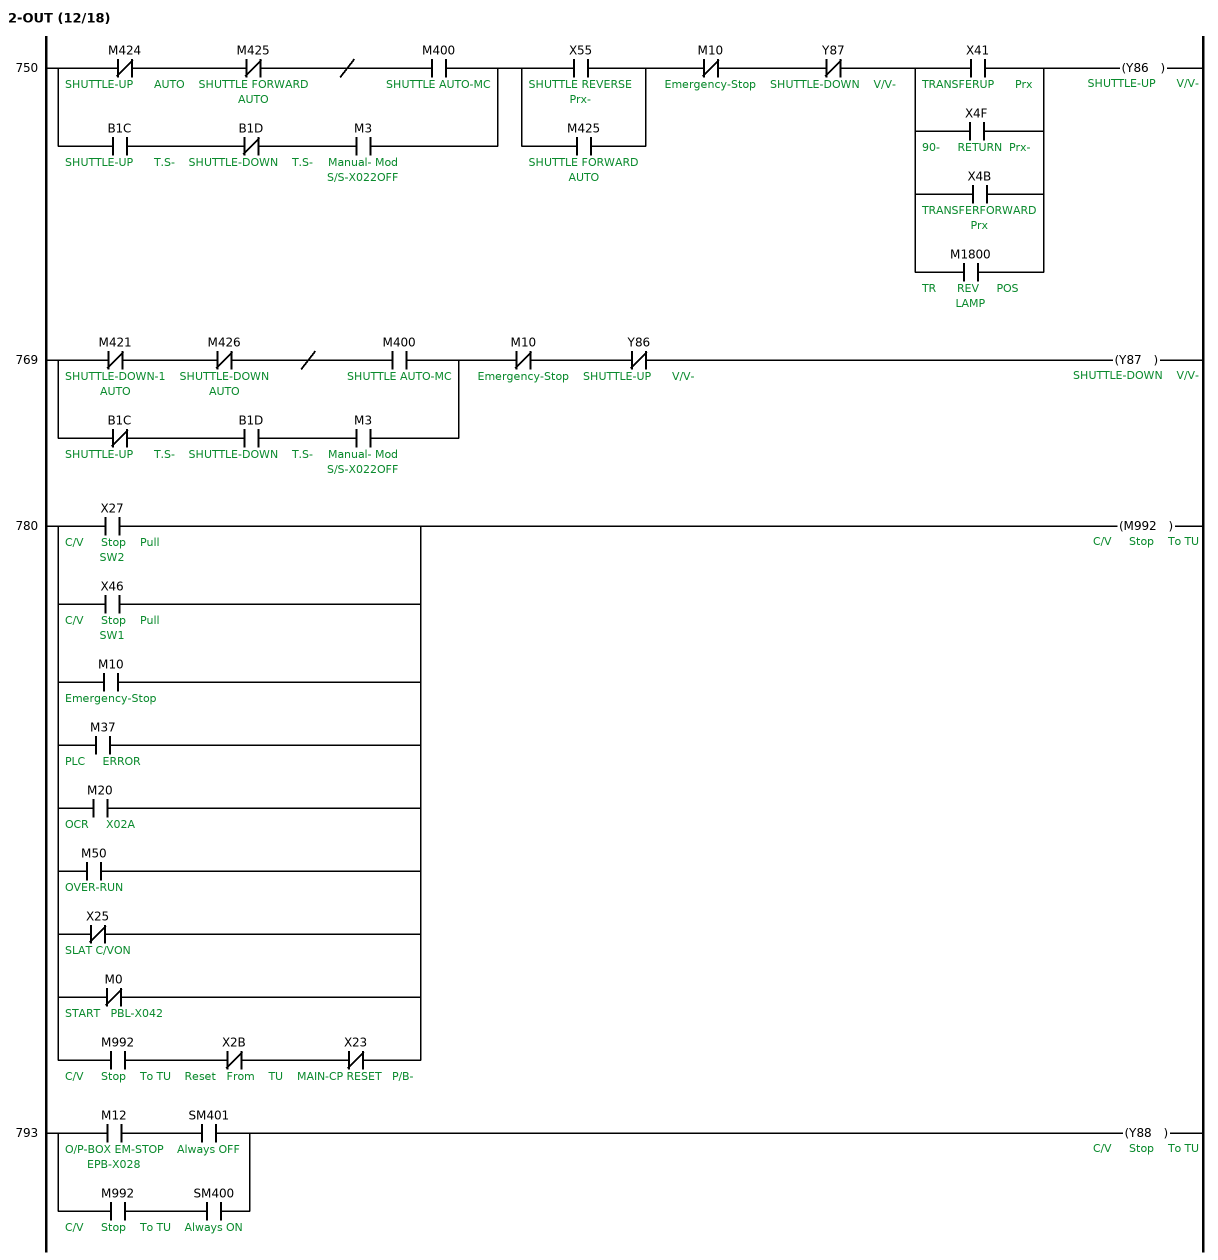
750   LDI     M424  ; SHUTTLE-UP      AUTO
      ANI     M425  ; SHUTTLE FORWARD AUTO
      INV
      AND     M400  ; SHUTTLE AUTO-MC
      LD      B1C  ; SHUTTLE-UP      T.S-
      ANI     B1D  ; SHUTTLE-DOWN    T.S-
      AND     M3  ; Manual- Mod     S/S-X022OFF
      ORB
      LD      X55  ; SHUTTLE REVERSE Prx-
      OR      M425  ; SHUTTLE FORWARD AUTO
      ANB
      ANI     M10  ; Emergency-Stop
      ANI     Y87  ; SHUTTLE-DOWN    V/V-
      LD      X41  ; TRANSFERUP      Prx
      OR      X4F  ; 90-     RETURN  Prx-
      OR      X4B  ; TRANSFERFORWARD Prx
      OR      M1800  ; TR      REV     POS     LAMP
      ANB
      OUT     Y86  ; SHUTTLE-UP      V/V-
769   LDI     M421  ; SHUTTLE-DOWN-1  AUTO
      ANI     M426  ; SHUTTLE-DOWN    AUTO
      INV
      AND     M400  ; SHUTTLE AUTO-MC
      LDI     B1C  ; SHUTTLE-UP      T.S-
      AND     B1D  ; SHUTTLE-DOWN    T.S-
      AND     M3  ; Manual- Mod     S/S-X022OFF
      ORB
      ANI     M10  ; Emergency-Stop
      ANI     Y86  ; SHUTTLE-UP      V/V-
      OUT     Y87  ; SHUTTLE-DOWN    V/V-
780   LD      X27  ; C/V     Stop    Pull    SW2
      OR      X46  ; C/V     Stop    Pull    SW1
      OR      M10  ; Emergency-Stop
      OR      M37  ; PLC     ERROR
      OR      M20  ; OCR     X02A
      OR      M50  ; OVER-RUN
      ORI     X25  ; SLAT C/VON
      ORI     M0  ; START   PBL-X042
      LD      M992  ; C/V     Stop    To TU
      ANI     X2B  ; Reset   From    TU
      ANI     X23  ; MAIN-CP RESET   P/B-
      ORB
      OUT     M992  ; C/V     Stop    To TU
793   LD      M12  ; O/P-BOX EM-STOP EPB-X028
      AND     SM401  ; Always OFF
      LD      M992  ; C/V     Stop    To TU
      AND     SM400  ; Always ON
      ORB
      OUT     Y88  ; C/V     Stop    To TU
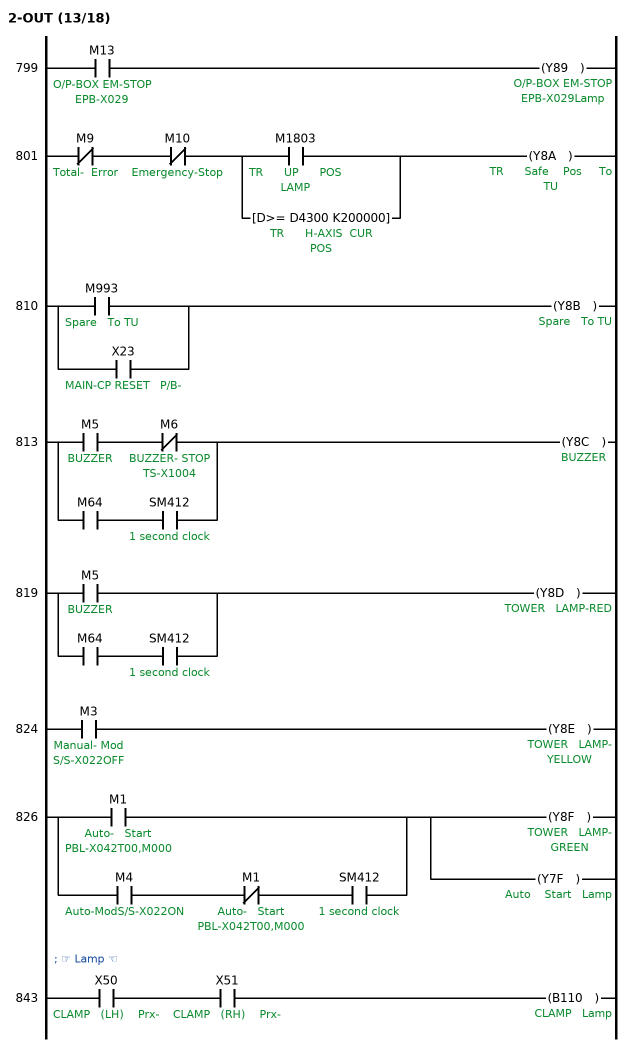
799   LD      M13  ; O/P-BOX EM-STOP EPB-X029
      OUT     Y89  ; O/P-BOX EM-STOP EPB-X029Lamp
801   LDI     M9  ; Total-  Error
      ANI     M10  ; Emergency-Stop
      LD      M1803  ; TR      UP      POS     LAMP
      ORD>=   D4300 K200000  ; TR      H-AXIS  CUR     POS
      ANB
      OUT     Y8A  ; TR      Safe    Pos     To TU
810   LD      M993  ; Spare   To TU
      OR      X23  ; MAIN-CP RESET   P/B-
      OUT     Y8B  ; Spare   To TU
813   LD      M5  ; BUZZER
      ANI     M6  ; BUZZER- STOP    TS-X1004
      LD      M64
      AND     SM412  ; 1 second clock
      ORB
      OUT     Y8C  ; BUZZER
819   LD      M5  ; BUZZER
      LD      M64
      AND     SM412  ; 1 second clock
      ORB
      OUT     Y8D  ; TOWER   LAMP-RED
824   LD      M3  ; Manual- Mod     S/S-X022OFF
      OUT     Y8E  ; TOWER   LAMP-   YELLOW
826   LD      M1  ; Auto-   Start   PBL-X042T00,M000
      LD      M4  ; Auto-ModS/S-X022ON
      ANI     M1  ; Auto-   Start   PBL-X042T00,M000
      AND     SM412  ; 1 second clock
      ORB
      OUT     Y8F  ; TOWER   LAMP-   GREEN
      OUT     Y7F  ; Auto    Start   Lamp
; ☞ Lamp ☜
843   LD      X50  ; CLAMP   (LH)    Prx-
      AND     X51  ; CLAMP   (RH)    Prx-
      OUT     B110  ; CLAMP   Lamp
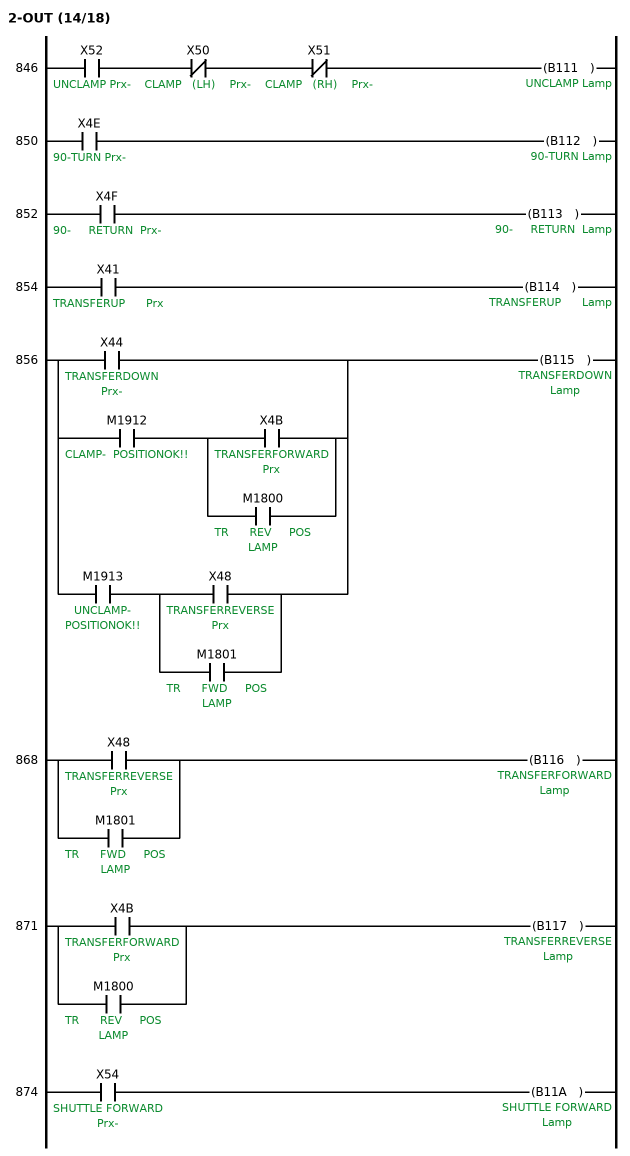
846   LD      X52  ; UNCLAMP Prx-
      ANI     X50  ; CLAMP   (LH)    Prx-
      ANI     X51  ; CLAMP   (RH)    Prx-
      OUT     B111  ; UNCLAMP Lamp
850   LD      X4E  ; 90-TURN Prx-
      OUT     B112  ; 90-TURN Lamp
852   LD      X4F  ; 90-     RETURN  Prx-
      OUT     B113  ; 90-     RETURN  Lamp
854   LD      X41  ; TRANSFERUP      Prx
      OUT     B114  ; TRANSFERUP      Lamp
856   LD      X44  ; TRANSFERDOWN    Prx-
      LD      M1912  ; CLAMP-  POSITIONOK!!
      LD      X4B  ; TRANSFERFORWARD Prx
      OR      M1800  ; TR      REV     POS     LAMP
      ANB
      ORB
      LD      M1913  ; UNCLAMP-POSITIONOK!!
      LD      X48  ; TRANSFERREVERSE Prx
      OR      M1801  ; TR      FWD     POS     LAMP
      ANB
      ORB
      OUT     B115  ; TRANSFERDOWN    Lamp
868   LD      X48  ; TRANSFERREVERSE Prx
      OR      M1801  ; TR      FWD     POS     LAMP
      OUT     B116  ; TRANSFERFORWARD Lamp
871   LD      X4B  ; TRANSFERFORWARD Prx
      OR      M1800  ; TR      REV     POS     LAMP
      OUT     B117  ; TRANSFERREVERSE Lamp
874   LD      X54  ; SHUTTLE FORWARD Prx-
      OUT     B11A  ; SHUTTLE FORWARD Lamp
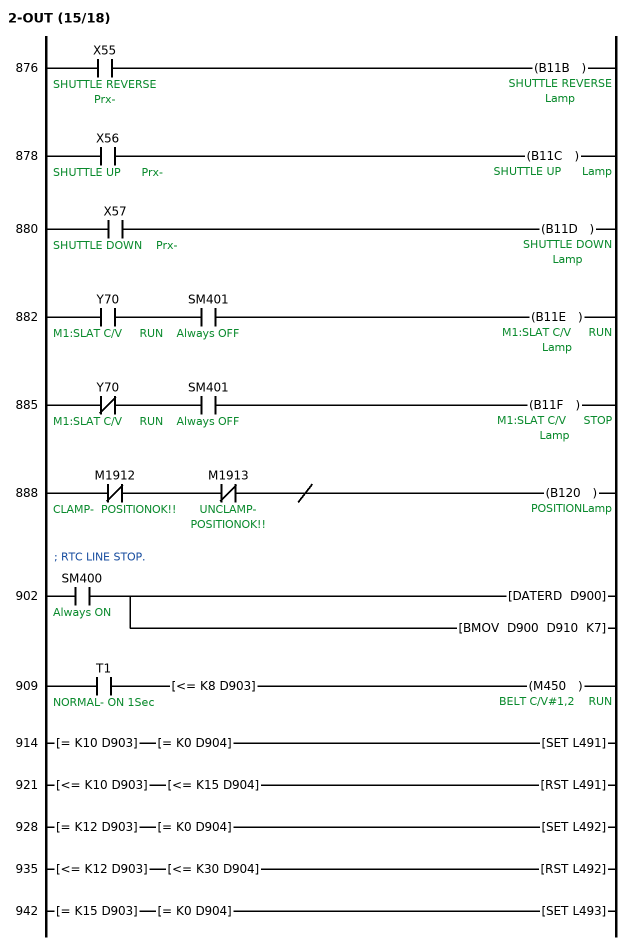
876   LD      X55  ; SHUTTLE REVERSE Prx-
      OUT     B11B  ; SHUTTLE REVERSE Lamp
878   LD      X56  ; SHUTTLE UP      Prx-
      OUT     B11C  ; SHUTTLE UP      Lamp
880   LD      X57  ; SHUTTLE DOWN    Prx-
      OUT     B11D  ; SHUTTLE DOWN    Lamp
882   LD      Y70  ; M1:SLAT C/V     RUN
      AND     SM401  ; Always OFF
      OUT     B11E  ; M1:SLAT C/V     RUN     Lamp
885   LDI     Y70  ; M1:SLAT C/V     RUN
      AND     SM401  ; Always OFF
      OUT     B11F  ; M1:SLAT C/V     STOP    Lamp
888   LDI     M1912  ; CLAMP-  POSITIONOK!!
      ANI     M1913  ; UNCLAMP-POSITIONOK!!
      INV
      OUT     B120  ; POSITIONLamp
; RTC LINE STOP.
902   LD      SM400  ; Always ON
      DATERD  D900
      BMOV    D900 D910 K7
909   LD      T1  ; NORMAL- ON 1Sec
      AND<=   K8 D903
      OUT     M450  ; BELT C/V#1,2    RUN
914   LD=     K10 D903
      AND=    K0 D904
      SET     L491
921   LD<=    K10 D903
      AND<=   K15 D904
      RST     L491
928   LD=     K12 D903
      AND=    K0 D904
      SET     L492
935   LD<=    K12 D903
      AND<=   K30 D904
      RST     L492
942   LD=     K15 D903
      AND=    K0 D904
      SET     L493
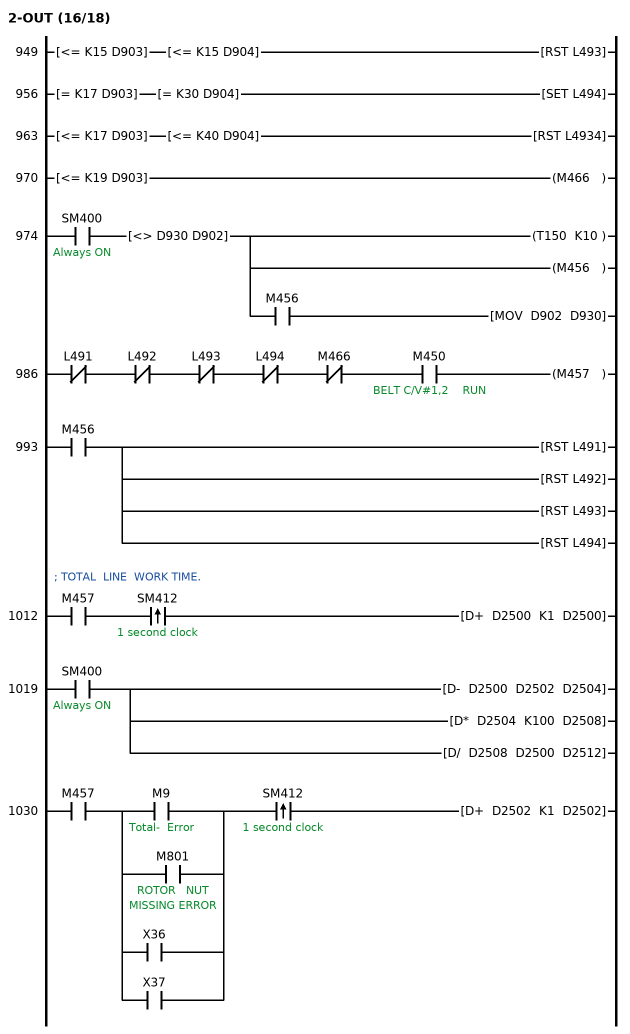
949   LD<=    K15 D903
      AND<=   K15 D904
      RST     L493
956   LD=     K17 D903
      AND=    K30 D904
      SET     L494
963   LD<=    K17 D903
      AND<=   K40 D904
      RST     L4934
970   LD<=    K19 D903
      OUT     M466
974   LD      SM400  ; Always ON
      AND<>   D930 D902
      OUT     T150 K10
      OUT     M456
      AND     M456
      MOV     D902 D930
986   LDI     L491
      ANI     L492
      ANI     L493
      ANI     L494
      ANI     M466
      AND     M450  ; BELT C/V#1,2    RUN
      OUT     M457
993   LD      M456
      RST     L491
      RST     L492
      RST     L493
      RST     L494
; TOTAL  LINE  WORK TIME.
1012  LD      M457
      ANDP    SM412  ; 1 second clock
      D+      D2500 K1 D2500
1019  LD      SM400  ; Always ON
      D-      D2500 D2502 D2504
      D*      D2504 K100 D2508
      D/      D2508 D2500 D2512
1030  LD      M457
      LD      M9  ; Total-  Error
      OR      M801  ; ROTOR   NUT     MISSING ERROR
      OR      X36
      OR      X37
      ANB
      ANDP    SM412  ; 1 second clock
      D+      D2502 K1 D2502
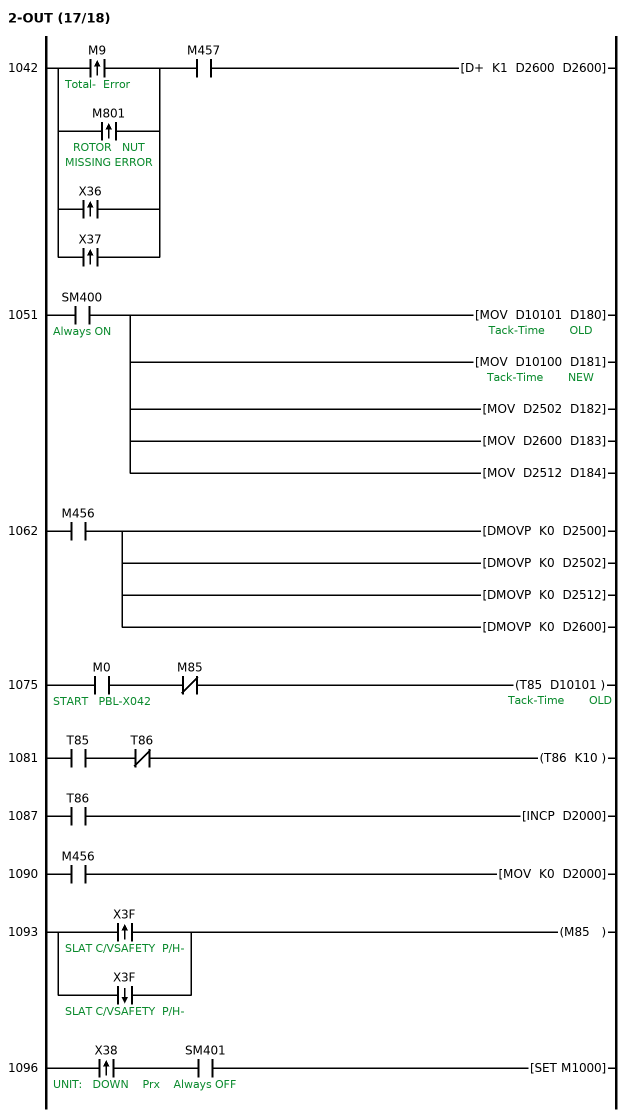
1042  LDP     M9  ; Total-  Error
      ORP     M801  ; ROTOR   NUT     MISSING ERROR
      ORP     X36
      ORP     X37
      AND     M457
      D+      K1 D2600 D2600
1051  LD      SM400  ; Always ON
      MOV     D10101 D180  ; Tack-Time       OLD
      MOV     D10100 D181  ; Tack-Time       NEW
      MOV     D2502 D182
      MOV     D2600 D183
      MOV     D2512 D184
1062  LD      M456
      DMOVP   K0 D2500
      DMOVP   K0 D2502
      DMOVP   K0 D2512
      DMOVP   K0 D2600
1075  LD      M0  ; START   PBL-X042
      ANI     M85
      OUT     T85 D10101  ; Tack-Time       OLD
1081  LD      T85
      ANI     T86
      OUT     T86 K10
1087  LD      T86
      INCP    D2000
1090  LD      M456
      MOV     K0 D2000
1093  LDP     X3F  ; SLAT C/VSAFETY  P/H-
      ORF     X3F  ; SLAT C/VSAFETY  P/H-
      OUT     M85
1096  LDP     X38  ; UNIT:   DOWN    Prx
      AND     SM401  ; Always OFF
      SET     M1000
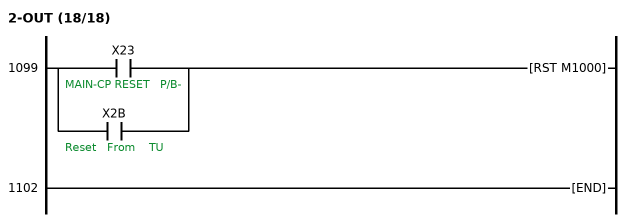
1099  LD      X23  ; MAIN-CP RESET   P/B-
      OR      X2B  ; Reset   From    TU
      RST     M1000
1102  END
END_PROGRAM

PROGRAM 3-ENCORD
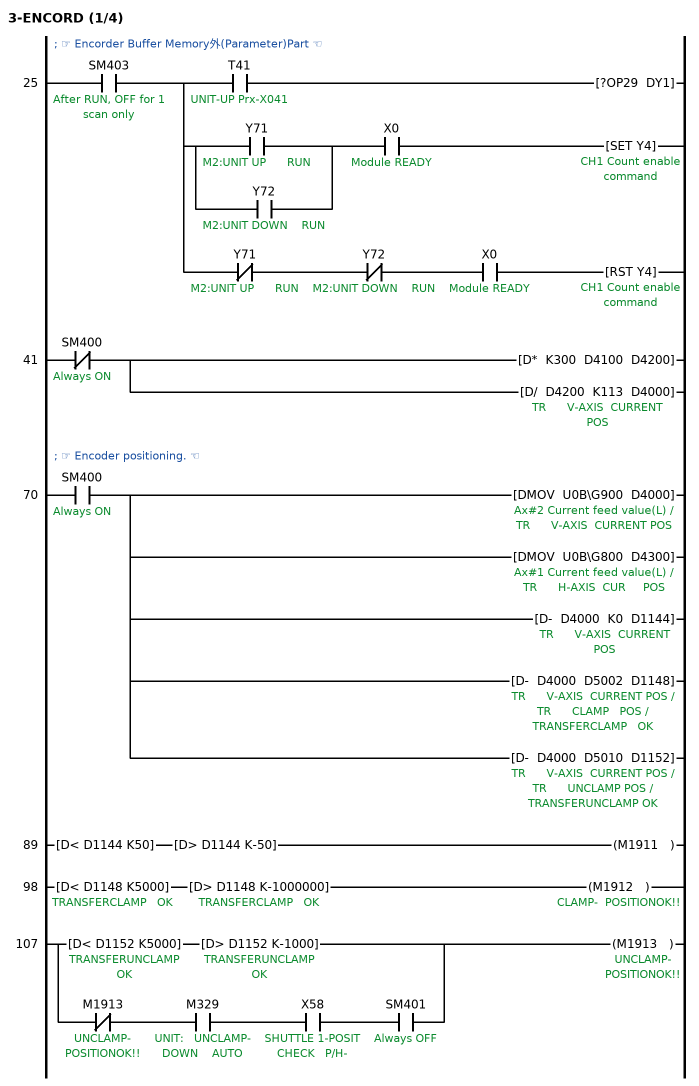
; ☞ Encorder Buffer Memory外(Parameter)Part ☜
25    LD      SM403  ; After RUN, OFF for 1 scan only
      MPS
      AND     T41  ; UNIT-UP Prx-X041
      ?OP29   DY1
      MRD
      LD      Y71  ; M2:UNIT UP      RUN
      OR      Y72  ; M2:UNIT DOWN    RUN
      ANB
      AND     X0  ; Module READY
      SET     Y4  ; CH1 Count enable command
      MPP
      ANI     Y71  ; M2:UNIT UP      RUN
      ANI     Y72  ; M2:UNIT DOWN    RUN
      AND     X0  ; Module READY
      RST     Y4  ; CH1 Count enable command
41    LDI     SM400  ; Always ON
      D*      K300 D4100 D4200
      D/      D4200 K113 D4000  ; TR      V-AXIS  CURRENT POS
; ☞ Encoder positioning. ☜
70    LD      SM400  ; Always ON
      DMOV    U0B\G900 D4000  ; Ax#2 Current feed value(L)
      DMOV    U0B\G800 D4300  ; Ax#1 Current feed value(L) / TR      H-AXIS  CUR     POS
      D-      D4000 K0 D1144
      D-      D4000 D5002 D1148  ; TR      CLAMP   POS / TRANSFERCLAMP   OK
      D-      D4000 D5010 D1152  ; TR      UNCLAMP POS / TRANSFERUNCLAMP OK
89    LDD<    D1144 K50
      ANDD>   D1144 K-50
      OUT     M1911
98    LDD<    D1148 K5000  ; TRANSFERCLAMP   OK
      ANDD>   D1148 K-1000000  ; TRANSFERCLAMP   OK
      OUT     M1912  ; CLAMP-  POSITIONOK!!
107   LDD<    D1152 K5000  ; TRANSFERUNCLAMP OK
      ANDD>   D1152 K-1000  ; TRANSFERUNCLAMP OK
      LDI     M1913  ; UNCLAMP-POSITIONOK!!
      AND     M329  ; UNIT:   UNCLAMP-DOWN    AUTO
      AND     X58  ; SHUTTLE 1-POSIT CHECK   P/H-
      AND     SM401  ; Always OFF
      ORB
      OUT     M1913  ; UNCLAMP-POSITIONOK!!
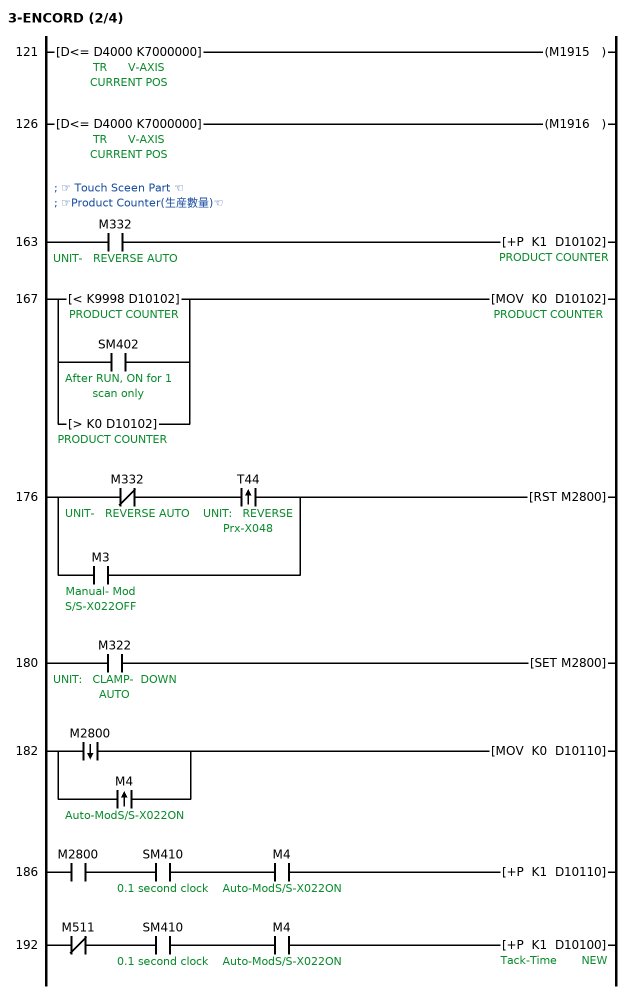
121   LDD<=   D4000 K7000000  ; TR      V-AXIS  CURRENT POS
      OUT     M1915
126   LDD<=   D4000 K7000000  ; TR      V-AXIS  CURRENT POS
      OUT     M1916
; ☞ Touch Sceen Part ☜
; ☞Product Counter(生産數量)☜
163   LD      M332  ; UNIT-   REVERSE AUTO
      +P      K1 D10102  ; PRODUCT COUNTER
167   LD<     K9998 D10102  ; PRODUCT COUNTER
      OR      SM402  ; After RUN, ON for 1 scan only
      OR>     K0 D10102  ; PRODUCT COUNTER
      MOV     K0 D10102
176   LDI     M332  ; UNIT-   REVERSE AUTO
      ANDP    T44  ; UNIT:   REVERSE Prx-X048
      OR      M3  ; Manual- Mod     S/S-X022OFF
      RST     M2800
180   LD      M322  ; UNIT:   CLAMP-  DOWN    AUTO
      SET     M2800
182   LDF     M2800
      ORP     M4  ; Auto-ModS/S-X022ON
      MOV     K0 D10110
186   LD      M2800
      AND     SM410  ; 0.1 second clock
      AND     M4  ; Auto-ModS/S-X022ON
      +P      K1 D10110
192   LDI     M511
      AND     SM410  ; 0.1 second clock
      AND     M4  ; Auto-ModS/S-X022ON
      +P      K1 D10100  ; Tack-Time       NEW
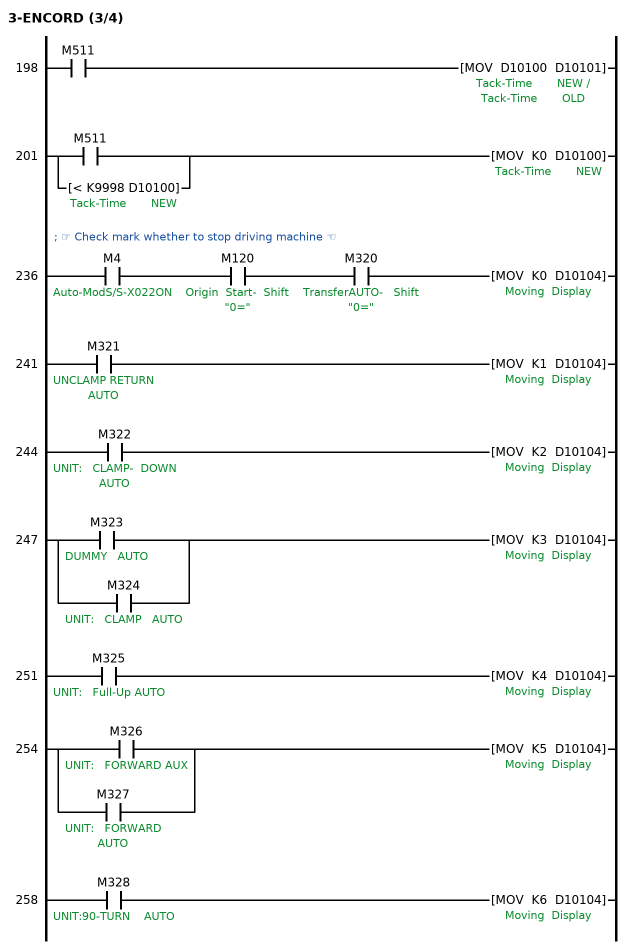
198   LD      M511
      MOV     D10100 D10101  ; Tack-Time       OLD
201   LD      M511
      OR<     K9998 D10100  ; Tack-Time       NEW
      MOV     K0 D10100
; ☞ Check mark whether to stop driving machine ☜
236   LD      M4  ; Auto-ModS/S-X022ON
      AND     M120  ; Origin  Start-  Shift   "0="
      AND     M320  ; TransferAUTO-   Shift   "0="
      MOV     K0 D10104  ; Moving  Display
241   LD      M321  ; UNCLAMP RETURN  AUTO
      MOV     K1 D10104
244   LD      M322  ; UNIT:   CLAMP-  DOWN    AUTO
      MOV     K2 D10104
247   LD      M323  ; DUMMY   AUTO
      OR      M324  ; UNIT:   CLAMP   AUTO
      MOV     K3 D10104
251   LD      M325  ; UNIT:   Full-Up AUTO
      MOV     K4 D10104
254   LD      M326  ; UNIT:   FORWARD AUX
      OR      M327  ; UNIT:   FORWARD AUTO
      MOV     K5 D10104
258   LD      M328  ; UNIT:90-TURN    AUTO
      MOV     K6 D10104
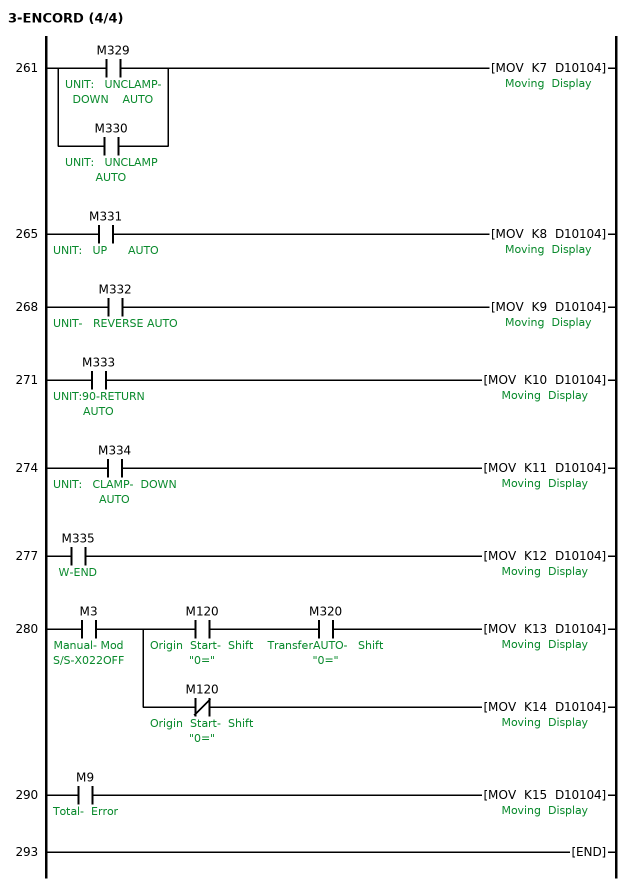
261   LD      M329  ; UNIT:   UNCLAMP-DOWN    AUTO
      OR      M330  ; UNIT:   UNCLAMP AUTO
      MOV     K7 D10104
265   LD      M331  ; UNIT:   UP      AUTO
      MOV     K8 D10104
268   LD      M332  ; UNIT-   REVERSE AUTO
      MOV     K9 D10104
271   LD      M333  ; UNIT:90-RETURN  AUTO
      MOV     K10 D10104
274   LD      M334  ; UNIT:   CLAMP-  DOWN    AUTO
      MOV     K11 D10104
277   LD      M335  ; W-END
      MOV     K12 D10104
280   LD      M3  ; Manual- Mod     S/S-X022OFF
      MPS
      AND     M120  ; Origin  Start-  Shift   "0="
      AND     M320  ; TransferAUTO-   Shift   "0="
      MOV     K13 D10104
      MPP
      ANI     M120  ; Origin  Start-  Shift   "0="
      MOV     K14 D10104
290   LD      M9  ; Total-  Error
      MOV     K15 D10104
293   END
END_PROGRAM

PROGRAM 4-MODEL
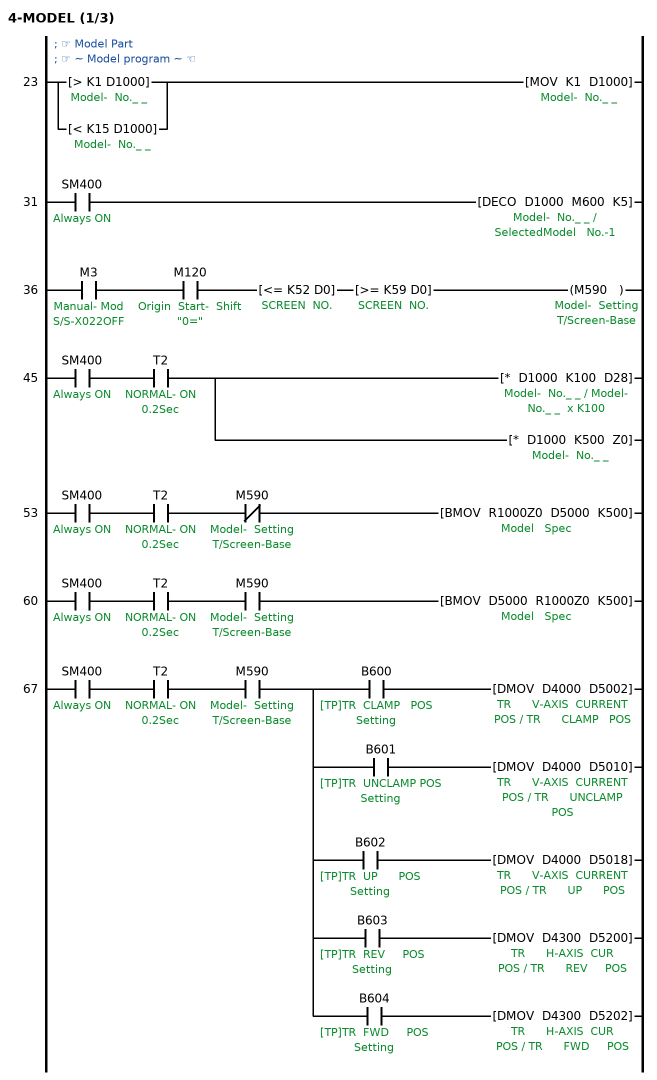
; ☞ Model Part
; ☞ ~ Model program ~ ☜
23    LD>     K1 D1000  ; Model-  No._ _
      OR<     K15 D1000  ; Model-  No._ _
      MOV     K1 D1000
31    LD      SM400  ; Always ON
      DECO    D1000 M600 K5  ; SelectedModel   No.-1
36    LD      M3  ; Manual- Mod     S/S-X022OFF
      AND     M120  ; Origin  Start-  Shift   "0="
      AND<=   K52 D0  ; SCREEN  NO.
      AND>=   K59 D0  ; SCREEN  NO.
      OUT     M590  ; Model-  Setting T/Screen-Base
45    LD      SM400  ; Always ON
      AND     T2  ; NORMAL- ON      0.2Sec
      *       D1000 K100 D28  ; Model-  No._ _  x K100
      *       D1000 K500 Z0
53    LD      SM400  ; Always ON
      AND     T2  ; NORMAL- ON      0.2Sec
      ANI     M590  ; Model-  Setting T/Screen-Base
      BMOV    R1000Z0 D5000 K500  ; Model   Spec
60    LD      SM400  ; Always ON
      AND     T2  ; NORMAL- ON      0.2Sec
      AND     M590  ; Model-  Setting T/Screen-Base
      BMOV    D5000 R1000Z0 K500
67    LD      SM400  ; Always ON
      AND     T2  ; NORMAL- ON      0.2Sec
      AND     M590  ; Model-  Setting T/Screen-Base
      MPS
      AND     B600  ; [TP]TR  CLAMP   POS     Setting
      DMOV    D4000 D5002  ; TR      V-AXIS  CURRENT POS / TR      CLAMP   POS
      MRD
      AND     B601  ; [TP]TR  UNCLAMP POS     Setting
      DMOV    D4000 D5010  ; TR      UNCLAMP POS
      MRD
      AND     B602  ; [TP]TR  UP      POS     Setting
      DMOV    D4000 D5018  ; TR      UP      POS
      MRD
      AND     B603  ; [TP]TR  REV     POS     Setting
      DMOV    D4300 D5200  ; TR      H-AXIS  CUR     POS / TR      REV     POS
      MPP
      AND     B604  ; [TP]TR  FWD     POS     Setting
      DMOV    D4300 D5202  ; TR      FWD     POS
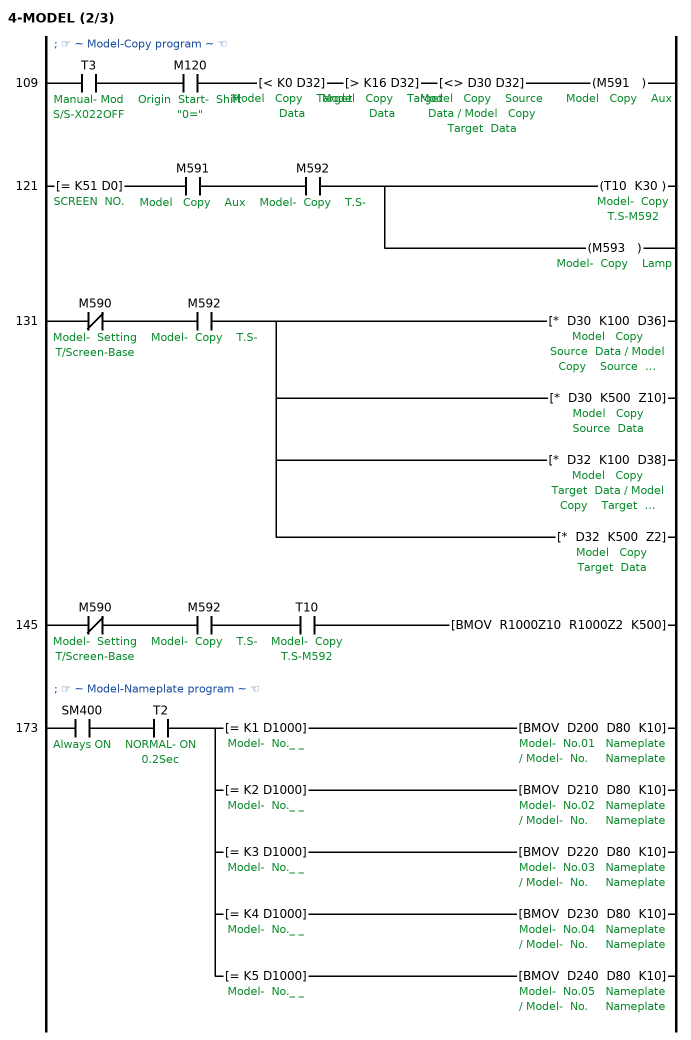
; ☞ ~ Model-Copy program ~ ☜
109   LD      T3  ; Manual- Mod     S/S-X022OFF
      AND     M120  ; Origin  Start-  Shift   "0="
      AND<    K0 D32  ; Model   Copy    Target  Data
      AND>    K16 D32  ; Model   Copy    Target  Data
      AND<>   D30 D32  ; Model   Copy    Source  Data / Model   Copy    Target  Data
      OUT     M591  ; Model   Copy    Aux
121   LD=     K51 D0  ; SCREEN  NO.
      AND     M591  ; Model   Copy    Aux
      AND     M592  ; Model-  Copy    T.S-
      OUT     T10 K30  ; Model-  Copy    T.S-M592
      OUT     M593  ; Model-  Copy    Lamp
131   LDI     M590  ; Model-  Setting T/Screen-Base
      AND     M592  ; Model-  Copy    T.S-
      *       D30 K100 D36  ; Model   Copy    Source  * K100
      *       D30 K500 Z10
      *       D32 K100 D38  ; Model   Copy    Target  * K100
      *       D32 K500 Z2
145   LDI     M590  ; Model-  Setting T/Screen-Base
      AND     M592  ; Model-  Copy    T.S-
      AND     T10  ; Model-  Copy    T.S-M592
      BMOV    R1000Z10 R1000Z2 K500
; ☞ ~ Model-Nameplate program ~ ☜
173   LD      SM400  ; Always ON
      AND     T2  ; NORMAL- ON      0.2Sec
      MPS
      AND=    K1 D1000  ; Model-  No._ _
      BMOV    D200 D80 K10  ; Model-  No.01   Nameplate / Model-  No.     Nameplate
      MRD
      AND=    K2 D1000  ; Model-  No._ _
      BMOV    D210 D80 K10  ; Model-  No.02   Nameplate
      MRD
      AND=    K3 D1000  ; Model-  No._ _
      BMOV    D220 D80 K10  ; Model-  No.03   Nameplate
      MRD
      AND=    K4 D1000  ; Model-  No._ _
      BMOV    D230 D80 K10  ; Model-  No.04   Nameplate
      MPP
      AND=    K5 D1000  ; Model-  No._ _
      BMOV    D240 D80 K10  ; Model-  No.05   Nameplate
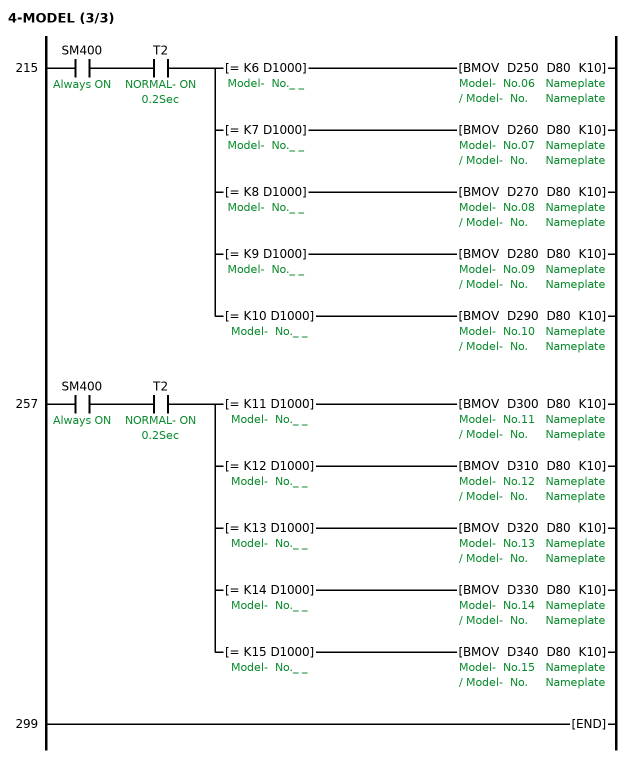
215   LD      SM400  ; Always ON
      AND     T2  ; NORMAL- ON      0.2Sec
      MPS
      AND=    K6 D1000  ; Model-  No._ _
      BMOV    D250 D80 K10  ; Model-  No.06   Nameplate
      MRD
      AND=    K7 D1000  ; Model-  No._ _
      BMOV    D260 D80 K10  ; Model-  No.07   Nameplate
      MRD
      AND=    K8 D1000  ; Model-  No._ _
      BMOV    D270 D80 K10  ; Model-  No.08   Nameplate
      MRD
      AND=    K9 D1000  ; Model-  No._ _
      BMOV    D280 D80 K10  ; Model-  No.09   Nameplate
      MPP
      AND=    K10 D1000  ; Model-  No._ _
      BMOV    D290 D80 K10  ; Model-  No.10   Nameplate
257   LD      SM400  ; Always ON
      AND     T2  ; NORMAL- ON      0.2Sec
      MPS
      AND=    K11 D1000  ; Model-  No._ _
      BMOV    D300 D80 K10  ; Model-  No.11   Nameplate
      MRD
      AND=    K12 D1000  ; Model-  No._ _
      BMOV    D310 D80 K10  ; Model-  No.12   Nameplate
      MRD
      AND=    K13 D1000  ; Model-  No._ _
      BMOV    D320 D80 K10  ; Model-  No.13   Nameplate
      MRD
      AND=    K14 D1000  ; Model-  No._ _
      BMOV    D330 D80 K10  ; Model-  No.14   Nameplate
      MPP
      AND=    K15 D1000  ; Model-  No._ _
      BMOV    D340 D80 K10  ; Model-  No.15   Nameplate
299   END
END_PROGRAM

PROGRAM 5-ERROR
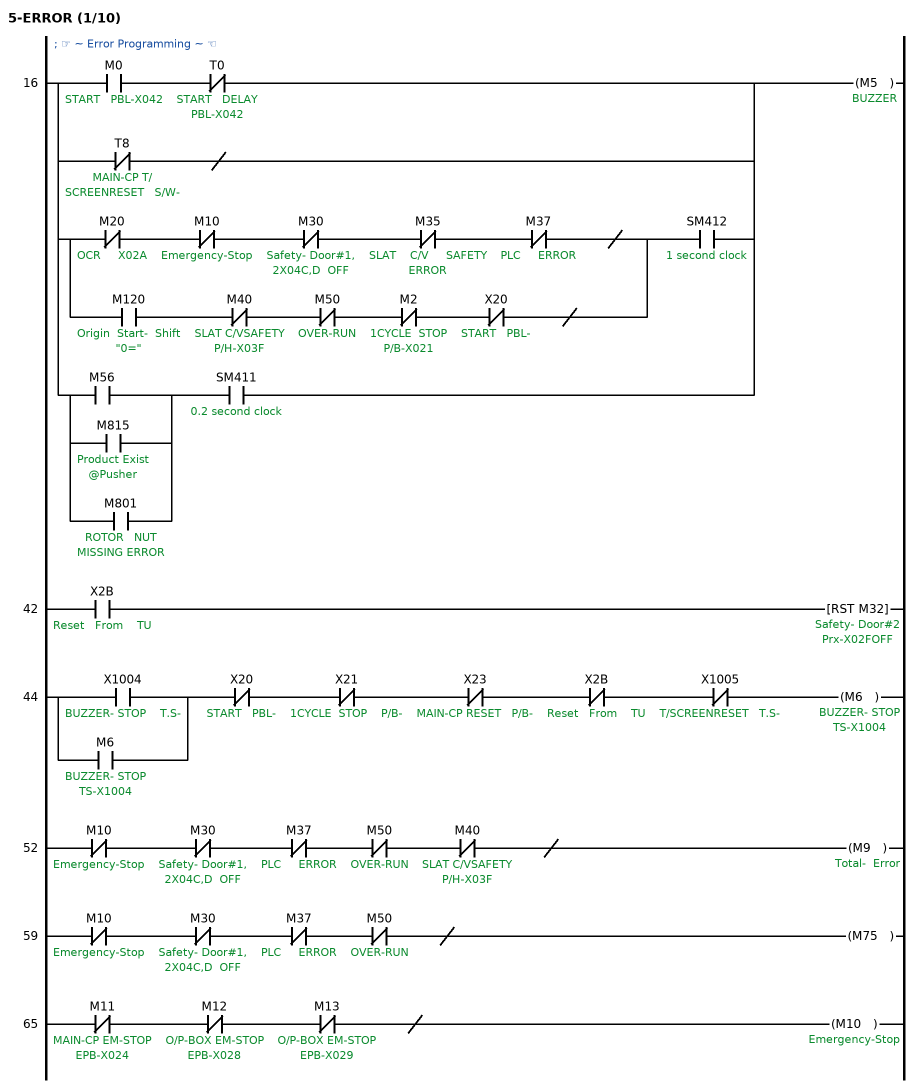
; ☞ ~ Error Programming ~ ☜
16    LD      M0  ; START   PBL-X042
      ANI     T0  ; START   DELAY   PBL-X042
      LDI     T8  ; MAIN-CP T/SCREENRESET   S/W-
      INV
      ORB
      LDI     M20  ; OCR     X02A
      ANI     M10  ; Emergency-Stop
      ANI     M30  ; Safety- Door#1,2X04C,D  OFF
      ANI     M35  ; SLAT    C/V     SAFETY  ERROR
      ANI     M37  ; PLC     ERROR
      INV
      LD      M120  ; Origin  Start-  Shift   "0="
      ANI     M40  ; SLAT C/VSAFETY  P/H-X03F
      ANI     M50  ; OVER-RUN
      ANI     M2  ; 1CYCLE  STOP    P/B-X021
      ANI     X20  ; START   PBL-
      INV
      ORB
      AND     SM412  ; 1 second clock
      ORB
      LD      M56
      OR      M815  ; Product Exist   @Pusher
      OR      M801  ; ROTOR   NUT     MISSING ERROR
      AND     SM411  ; 0.2 second clock
      ORB
      OUT     M5  ; BUZZER
42    LD      X2B  ; Reset   From    TU
      RST     M32  ; Safety- Door#2  Prx-X02FOFF
44    LD      X1004  ; BUZZER- STOP    T.S-
      OR      M6  ; BUZZER- STOP    TS-X1004
      ANI     X20  ; START   PBL-
      ANI     X21  ; 1CYCLE  STOP    P/B-
      ANI     X23  ; MAIN-CP RESET   P/B-
      ANI     X2B  ; Reset   From    TU
      ANI     X1005  ; T/SCREENRESET   T.S-
      OUT     M6  ; BUZZER- STOP    TS-X1004
52    LDI     M10  ; Emergency-Stop
      ANI     M30  ; Safety- Door#1,2X04C,D  OFF
      ANI     M37  ; PLC     ERROR
      ANI     M50  ; OVER-RUN
      ANI     M40  ; SLAT C/VSAFETY  P/H-X03F
      INV
      OUT     M9  ; Total-  Error
59    LDI     M10  ; Emergency-Stop
      ANI     M30  ; Safety- Door#1,2X04C,D  OFF
      ANI     M37  ; PLC     ERROR
      ANI     M50  ; OVER-RUN
      INV
      OUT     M75
65    LDI     M11  ; MAIN-CP EM-STOP EPB-X024
      ANI     M12  ; O/P-BOX EM-STOP EPB-X028
      ANI     M13  ; O/P-BOX EM-STOP EPB-X029
      INV
      OUT     M10  ; Emergency-Stop
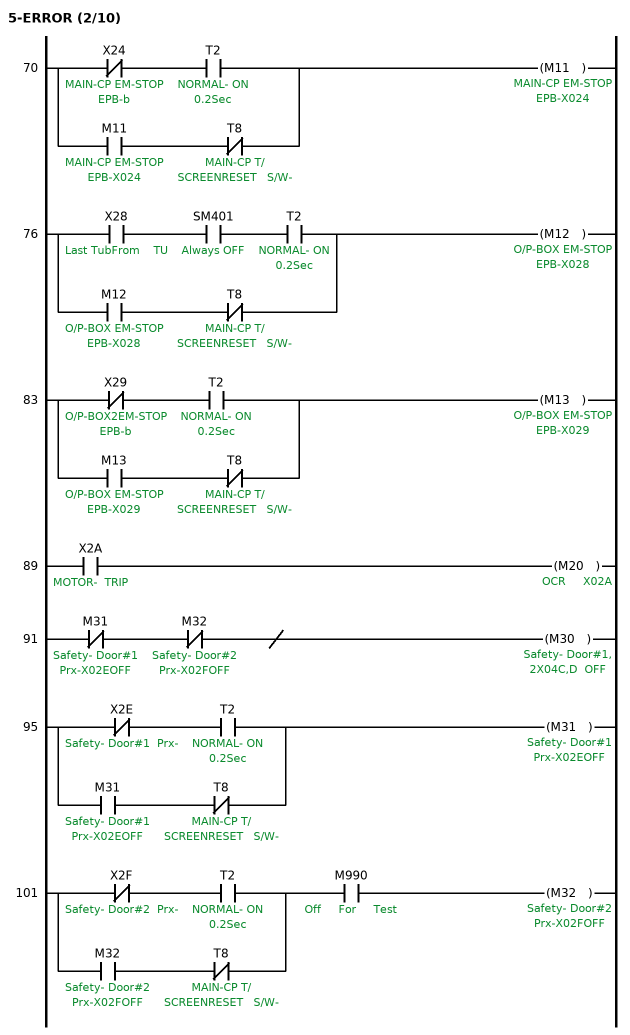
70    LDI     X24  ; MAIN-CP EM-STOP EPB-b
      AND     T2  ; NORMAL- ON      0.2Sec
      LD      M11  ; MAIN-CP EM-STOP EPB-X024
      ANI     T8  ; MAIN-CP T/SCREENRESET   S/W-
      ORB
      OUT     M11  ; MAIN-CP EM-STOP EPB-X024
76    LD      X28  ; Last TubFrom    TU
      AND     SM401  ; Always OFF
      AND     T2  ; NORMAL- ON      0.2Sec
      LD      M12  ; O/P-BOX EM-STOP EPB-X028
      ANI     T8  ; MAIN-CP T/SCREENRESET   S/W-
      ORB
      OUT     M12  ; O/P-BOX EM-STOP EPB-X028
83    LDI     X29  ; O/P-BOX2EM-STOP EPB-b
      AND     T2  ; NORMAL- ON      0.2Sec
      LD      M13  ; O/P-BOX EM-STOP EPB-X029
      ANI     T8  ; MAIN-CP T/SCREENRESET   S/W-
      ORB
      OUT     M13  ; O/P-BOX EM-STOP EPB-X029
89    LD      X2A  ; MOTOR-  TRIP
      OUT     M20  ; OCR     X02A
91    LDI     M31  ; Safety- Door#1  Prx-X02EOFF
      ANI     M32  ; Safety- Door#2  Prx-X02FOFF
      INV
      OUT     M30  ; Safety- Door#1,2X04C,D  OFF
95    LDI     X2E  ; Safety- Door#1  Prx-
      AND     T2  ; NORMAL- ON      0.2Sec
      LD      M31  ; Safety- Door#1  Prx-X02EOFF
      ANI     T8  ; MAIN-CP T/SCREENRESET   S/W-
      ORB
      OUT     M31  ; Safety- Door#1  Prx-X02EOFF
101   LDI     X2F  ; Safety- Door#2  Prx-
      AND     T2  ; NORMAL- ON      0.2Sec
      LD      M32  ; Safety- Door#2  Prx-X02FOFF
      ANI     T8  ; MAIN-CP T/SCREENRESET   S/W-
      ORB
      AND     M990  ; Off     For     Test
      OUT     M32  ; Safety- Door#2  Prx-X02FOFF
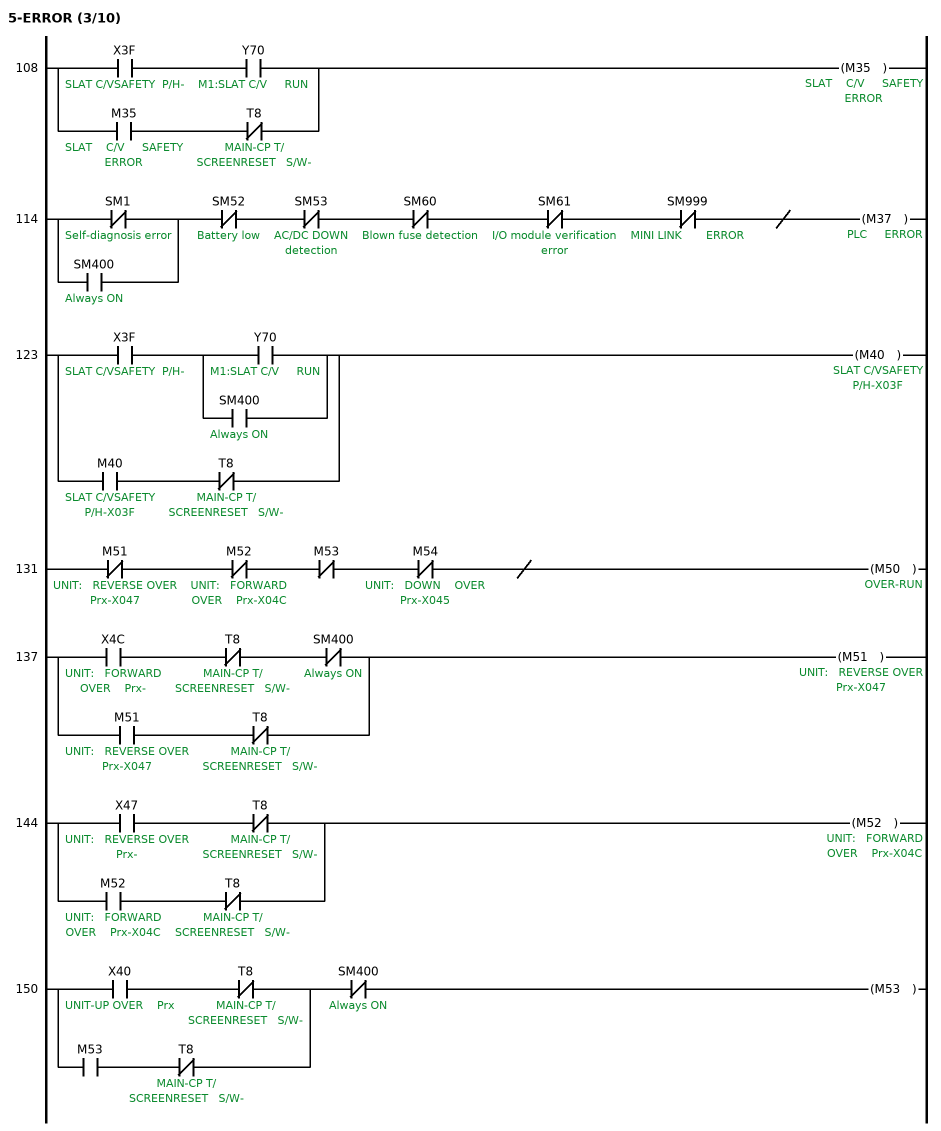
108   LD      X3F  ; SLAT C/VSAFETY  P/H-
      AND     Y70  ; M1:SLAT C/V     RUN
      LD      M35  ; SLAT    C/V     SAFETY  ERROR
      ANI     T8  ; MAIN-CP T/SCREENRESET   S/W-
      ORB
      OUT     M35  ; SLAT    C/V     SAFETY  ERROR
114   LDI     SM1  ; Self-diagnosis error
      OR      SM400  ; Always ON
      ANI     SM52  ; Battery low
      ANI     SM53  ; AC/DC DOWN detection
      ANI     SM60  ; Blown fuse detection
      ANI     SM61  ; I/O module verification error
      ANI     SM999  ; MINI LINK       ERROR
      INV
      OUT     M37  ; PLC     ERROR
123   LD      X3F  ; SLAT C/VSAFETY  P/H-
      LD      Y70  ; M1:SLAT C/V     RUN
      OR      SM400  ; Always ON
      ANB
      LD      M40  ; SLAT C/VSAFETY  P/H-X03F
      ANI     T8  ; MAIN-CP T/SCREENRESET   S/W-
      ORB
      OUT     M40  ; SLAT C/VSAFETY  P/H-X03F
131   LDI     M51  ; UNIT:   REVERSE OVER    Prx-X047
      ANI     M52  ; UNIT:   FORWARD OVER    Prx-X04C
      ANI     M53
      ANI     M54  ; UNIT:   DOWN    OVER    Prx-X045
      INV
      OUT     M50  ; OVER-RUN
137   LD      X4C  ; UNIT:   FORWARD OVER    Prx-
      ANI     T8  ; MAIN-CP T/SCREENRESET   S/W-
      ANI     SM400  ; Always ON
      LD      M51  ; UNIT:   REVERSE OVER    Prx-X047
      ANI     T8  ; MAIN-CP T/SCREENRESET   S/W-
      ORB
      OUT     M51  ; UNIT:   REVERSE OVER    Prx-X047
144   LD      X47  ; UNIT:   REVERSE OVER    Prx-
      ANI     T8  ; MAIN-CP T/SCREENRESET   S/W-
      LD      M52  ; UNIT:   FORWARD OVER    Prx-X04C
      ANI     T8  ; MAIN-CP T/SCREENRESET   S/W-
      ORB
      OUT     M52  ; UNIT:   FORWARD OVER    Prx-X04C
150   LD      X40  ; UNIT-UP OVER    Prx
      ANI     T8  ; MAIN-CP T/SCREENRESET   S/W-
      LD      M53
      ANI     T8  ; MAIN-CP T/SCREENRESET   S/W-
      ORB
      ANI     SM400  ; Always ON
      OUT     M53
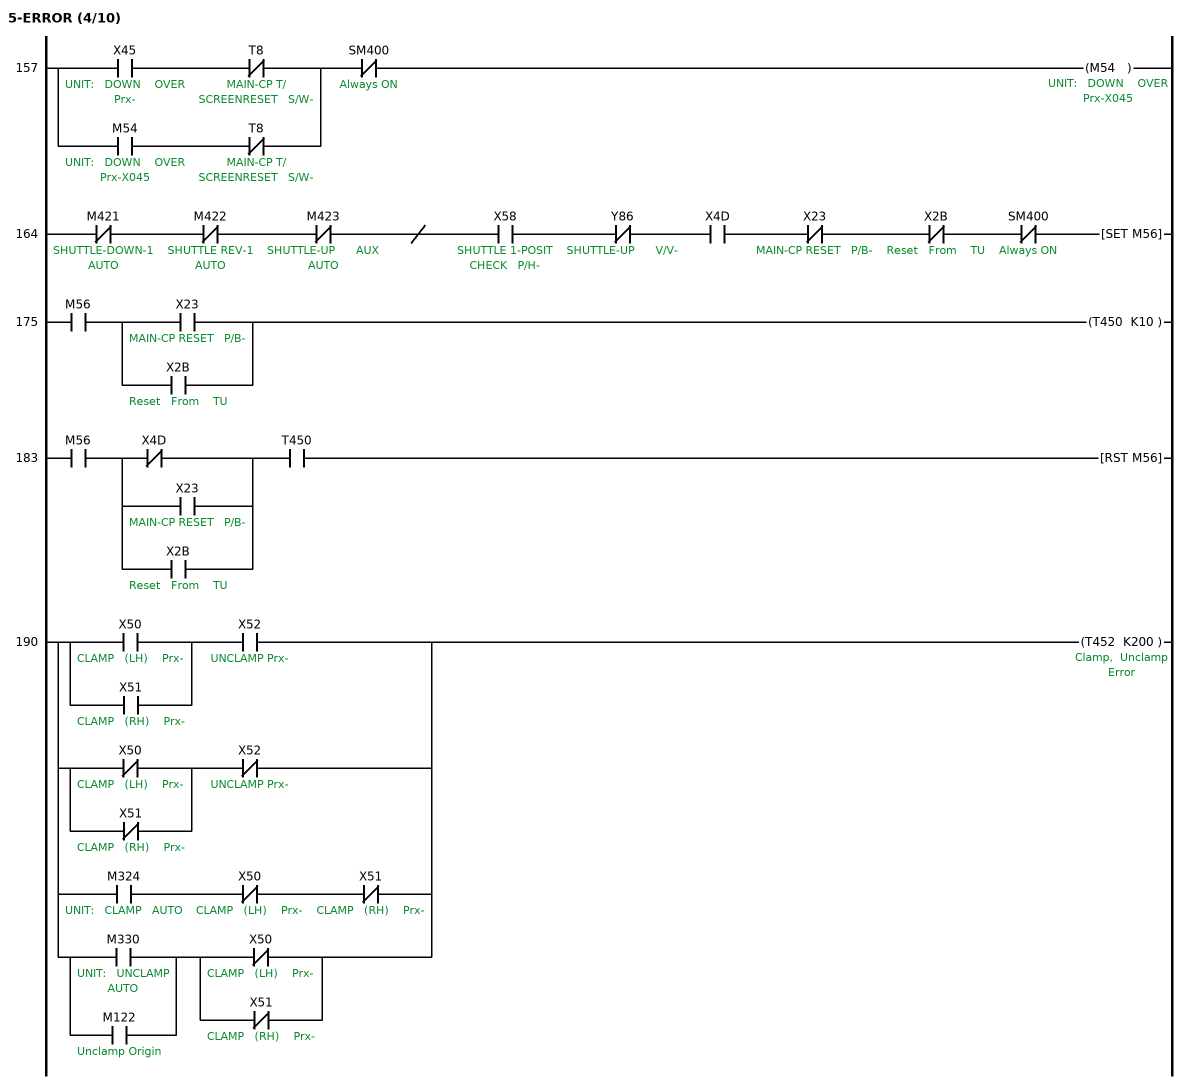
157   LD      X45  ; UNIT:   DOWN    OVER    Prx-
      ANI     T8  ; MAIN-CP T/SCREENRESET   S/W-
      LD      M54  ; UNIT:   DOWN    OVER    Prx-X045
      ANI     T8  ; MAIN-CP T/SCREENRESET   S/W-
      ORB
      ANI     SM400  ; Always ON
      OUT     M54  ; UNIT:   DOWN    OVER    Prx-X045
164   LDI     M421  ; SHUTTLE-DOWN-1  AUTO
      ANI     M422  ; SHUTTLE REV-1   AUTO
      ANI     M423  ; SHUTTLE-UP      AUX     AUTO
      INV
      AND     X58  ; SHUTTLE 1-POSIT CHECK   P/H-
      ANI     Y86  ; SHUTTLE-UP      V/V-
      AND     X4D
      ANI     X23  ; MAIN-CP RESET   P/B-
      ANI     X2B  ; Reset   From    TU
      ANI     SM400  ; Always ON
      SET     M56
175   LD      M56
      LD      X23  ; MAIN-CP RESET   P/B-
      OR      X2B  ; Reset   From    TU
      ANB
      OUT     T450 K10
183   LD      M56
      LDI     X4D
      OR      X23  ; MAIN-CP RESET   P/B-
      OR      X2B  ; Reset   From    TU
      ANB
      AND     T450
      RST     M56
190   LD      X50  ; CLAMP   (LH)    Prx-
      OR      X51  ; CLAMP   (RH)    Prx-
      AND     X52  ; UNCLAMP Prx-
      LDI     X50  ; CLAMP   (LH)    Prx-
      ORI     X51  ; CLAMP   (RH)    Prx-
      ANI     X52  ; UNCLAMP Prx-
      ORB
      LD      M324  ; UNIT:   CLAMP   AUTO
      ANI     X50  ; CLAMP   (LH)    Prx-
      ANI     X51  ; CLAMP   (RH)    Prx-
      ORB
      LD      M330  ; UNIT:   UNCLAMP AUTO
      OR      M122  ; Unclamp Origin
      LDI     X50  ; CLAMP   (LH)    Prx-
      ORI     X51  ; CLAMP   (RH)    Prx-
      ANB
      ORB
      OUT     T452 K200  ; Clamp,  Unclamp Error
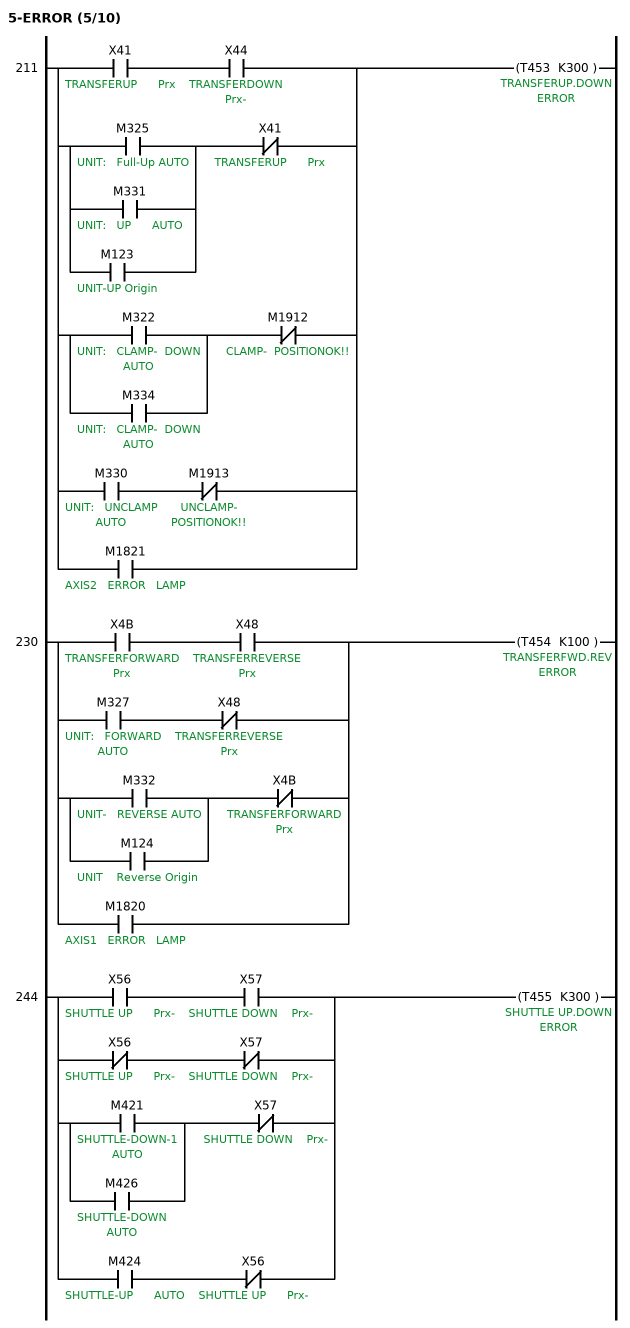
211   LD      X41  ; TRANSFERUP      Prx
      AND     X44  ; TRANSFERDOWN    Prx-
      LD      M325  ; UNIT:   Full-Up AUTO
      OR      M331  ; UNIT:   UP      AUTO
      OR      M123  ; UNIT-UP Origin
      ANI     X41  ; TRANSFERUP      Prx
      ORB
      LD      M322  ; UNIT:   CLAMP-  DOWN    AUTO
      OR      M334  ; UNIT:   CLAMP-  DOWN    AUTO
      ANI     M1912  ; CLAMP-  POSITIONOK!!
      ORB
      LD      M330  ; UNIT:   UNCLAMP AUTO
      ANI     M1913  ; UNCLAMP-POSITIONOK!!
      ORB
      OR      M1821  ; AXIS2   ERROR   LAMP
      OUT     T453 K300  ; TRANSFERUP.DOWN ERROR
230   LD      X4B  ; TRANSFERFORWARD Prx
      AND     X48  ; TRANSFERREVERSE Prx
      LD      M327  ; UNIT:   FORWARD AUTO
      ANI     X48  ; TRANSFERREVERSE Prx
      ORB
      LD      M332  ; UNIT-   REVERSE AUTO
      OR      M124  ; UNIT    Reverse Origin
      ANI     X4B  ; TRANSFERFORWARD Prx
      ORB
      OR      M1820  ; AXIS1   ERROR   LAMP
      OUT     T454 K100  ; TRANSFERFWD.REV ERROR
244   LD      X56  ; SHUTTLE UP      Prx-
      AND     X57  ; SHUTTLE DOWN    Prx-
      LDI     X56  ; SHUTTLE UP      Prx-
      ANI     X57  ; SHUTTLE DOWN    Prx-
      ORB
      LD      M421  ; SHUTTLE-DOWN-1  AUTO
      OR      M426  ; SHUTTLE-DOWN    AUTO
      ANI     X57  ; SHUTTLE DOWN    Prx-
      ORB
      LD      M424  ; SHUTTLE-UP      AUTO
      ANI     X56  ; SHUTTLE UP      Prx-
      ORB
      OUT     T455 K300  ; SHUTTLE UP.DOWN ERROR
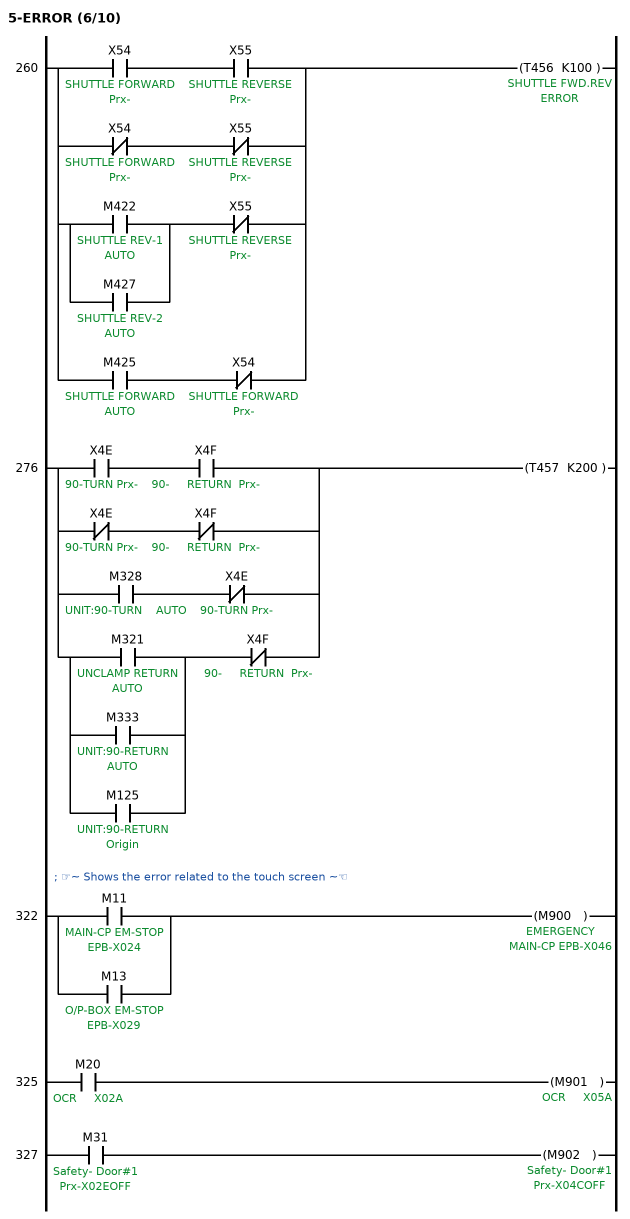
260   LD      X54  ; SHUTTLE FORWARD Prx-
      AND     X55  ; SHUTTLE REVERSE Prx-
      LDI     X54  ; SHUTTLE FORWARD Prx-
      ANI     X55  ; SHUTTLE REVERSE Prx-
      ORB
      LD      M422  ; SHUTTLE REV-1   AUTO
      OR      M427  ; SHUTTLE REV-2   AUTO
      ANI     X55  ; SHUTTLE REVERSE Prx-
      ORB
      LD      M425  ; SHUTTLE FORWARD AUTO
      ANI     X54  ; SHUTTLE FORWARD Prx-
      ORB
      OUT     T456 K100  ; SHUTTLE FWD.REV ERROR
276   LD      X4E  ; 90-TURN Prx-
      AND     X4F  ; 90-     RETURN  Prx-
      LDI     X4E  ; 90-TURN Prx-
      ANI     X4F  ; 90-     RETURN  Prx-
      ORB
      LD      M328  ; UNIT:90-TURN    AUTO
      ANI     X4E  ; 90-TURN Prx-
      ORB
      LD      M321  ; UNCLAMP RETURN  AUTO
      OR      M333  ; UNIT:90-RETURN  AUTO
      OR      M125  ; UNIT:90-RETURN  Origin
      ANI     X4F  ; 90-     RETURN  Prx-
      ORB
      OUT     T457 K200
; ☞~ Shows the error related to the touch screen ~☜
322   LD      M11  ; MAIN-CP EM-STOP EPB-X024
      OR      M13  ; O/P-BOX EM-STOP EPB-X029
      OUT     M900  ; EMERGENCY       MAIN-CP EPB-X046
325   LD      M20  ; OCR     X02A
      OUT     M901  ; OCR     X05A
327   LD      M31  ; Safety- Door#1  Prx-X02EOFF
      OUT     M902  ; Safety- Door#1  Prx-X04COFF
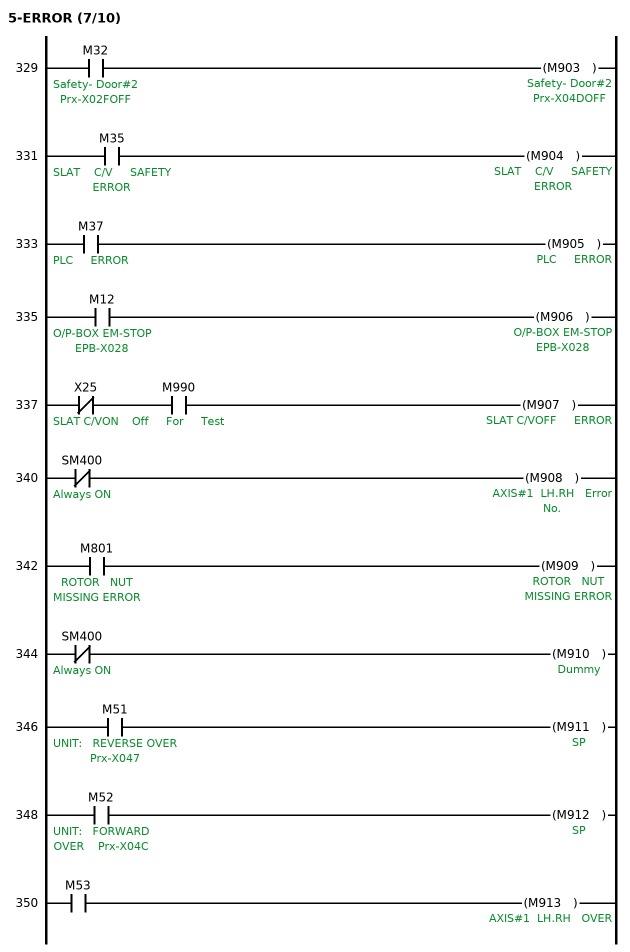
329   LD      M32  ; Safety- Door#2  Prx-X02FOFF
      OUT     M903  ; Safety- Door#2  Prx-X04DOFF
331   LD      M35  ; SLAT    C/V     SAFETY  ERROR
      OUT     M904  ; SLAT    C/V     SAFETY  ERROR
333   LD      M37  ; PLC     ERROR
      OUT     M905  ; PLC     ERROR
335   LD      M12  ; O/P-BOX EM-STOP EPB-X028
      OUT     M906  ; O/P-BOX EM-STOP EPB-X028
337   LDI     X25  ; SLAT C/VON
      AND     M990  ; Off     For     Test
      OUT     M907  ; SLAT C/VOFF     ERROR
340   LDI     SM400  ; Always ON
      OUT     M908  ; AXIS#1  LH.RH   Error   No.
342   LD      M801  ; ROTOR   NUT     MISSING ERROR
      OUT     M909  ; ROTOR   NUT     MISSING ERROR
344   LDI     SM400  ; Always ON
      OUT     M910  ; Dummy
346   LD      M51  ; UNIT:   REVERSE OVER    Prx-X047
      OUT     M911  ; SP
348   LD      M52  ; UNIT:   FORWARD OVER    Prx-X04C
      OUT     M912  ; SP
350   LD      M53
      OUT     M913  ; AXIS#1  LH.RH   OVER
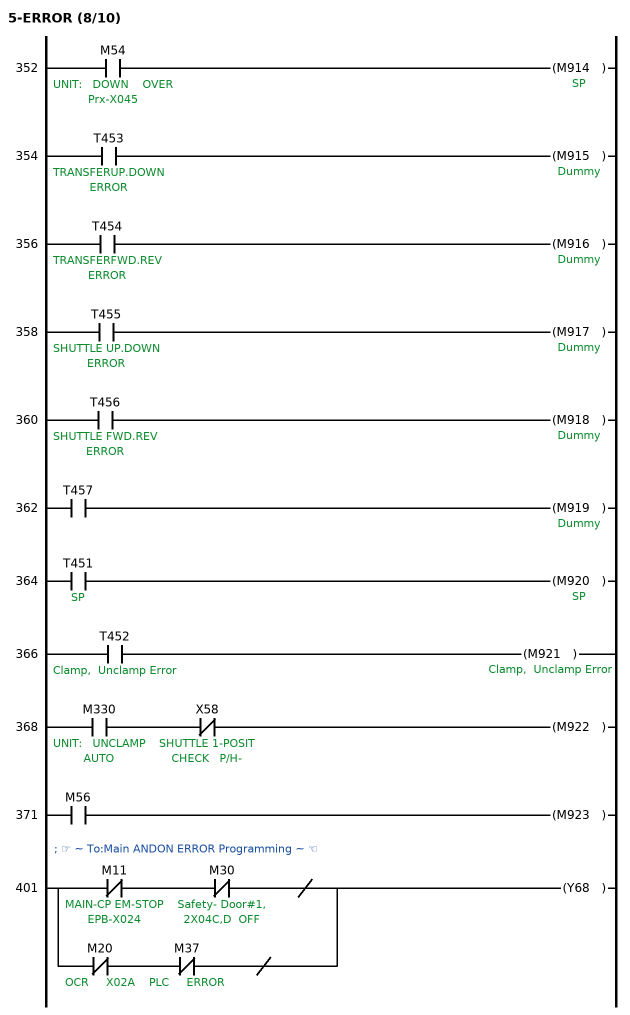
352   LD      M54  ; UNIT:   DOWN    OVER    Prx-X045
      OUT     M914  ; SP
354   LD      T453  ; TRANSFERUP.DOWN ERROR
      OUT     M915  ; Dummy
356   LD      T454  ; TRANSFERFWD.REV ERROR
      OUT     M916  ; Dummy
358   LD      T455  ; SHUTTLE UP.DOWN ERROR
      OUT     M917  ; Dummy
360   LD      T456  ; SHUTTLE FWD.REV ERROR
      OUT     M918  ; Dummy
362   LD      T457
      OUT     M919  ; Dummy
364   LD      T451  ; SP
      OUT     M920  ; SP
366   LD      T452  ; Clamp,  Unclamp Error
      OUT     M921  ; Clamp,  Unclamp Error
368   LD      M330  ; UNIT:   UNCLAMP AUTO
      ANI     X58  ; SHUTTLE 1-POSIT CHECK   P/H-
      OUT     M922
371   LD      M56
      OUT     M923
; ☞ ~ To:Main ANDON ERROR Programming ~ ☜
401   LDI     M11  ; MAIN-CP EM-STOP EPB-X024
      ANI     M30  ; Safety- Door#1,2X04C,D  OFF
      INV
      LDI     M20  ; OCR     X02A
      ANI     M37  ; PLC     ERROR
      INV
      ORB
      OUT     Y68
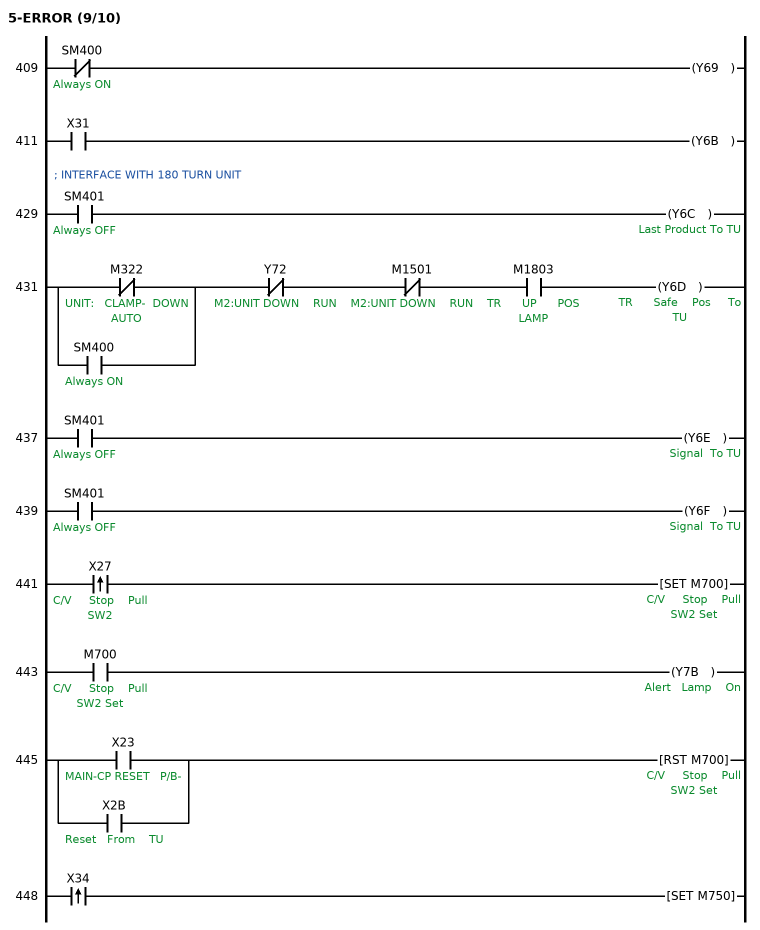
409   LDI     SM400  ; Always ON
      OUT     Y69
411   LD      X31
      OUT     Y6B
; INTERFACE WITH 180 TURN UNIT
429   LD      SM401  ; Always OFF
      OUT     Y6C  ; Last Product To TU
431   LDI     M322  ; UNIT:   CLAMP-  DOWN    AUTO
      OR      SM400  ; Always ON
      ANI     Y72  ; M2:UNIT DOWN    RUN
      ANI     M1501  ; M2:UNIT DOWN    RUN
      AND     M1803  ; TR      UP      POS     LAMP
      OUT     Y6D  ; TR      Safe    Pos     To TU
437   LD      SM401  ; Always OFF
      OUT     Y6E  ; Signal  To TU
439   LD      SM401  ; Always OFF
      OUT     Y6F  ; Signal  To TU
441   LDP     X27  ; C/V     Stop    Pull    SW2
      SET     M700  ; C/V     Stop    Pull    SW2 Set
443   LD      M700  ; C/V     Stop    Pull    SW2 Set
      OUT     Y7B  ; Alert   Lamp    On
445   LD      X23  ; MAIN-CP RESET   P/B-
      OR      X2B  ; Reset   From    TU
      RST     M700  ; C/V     Stop    Pull    SW2 Set
448   LDP     X34
      SET     M750
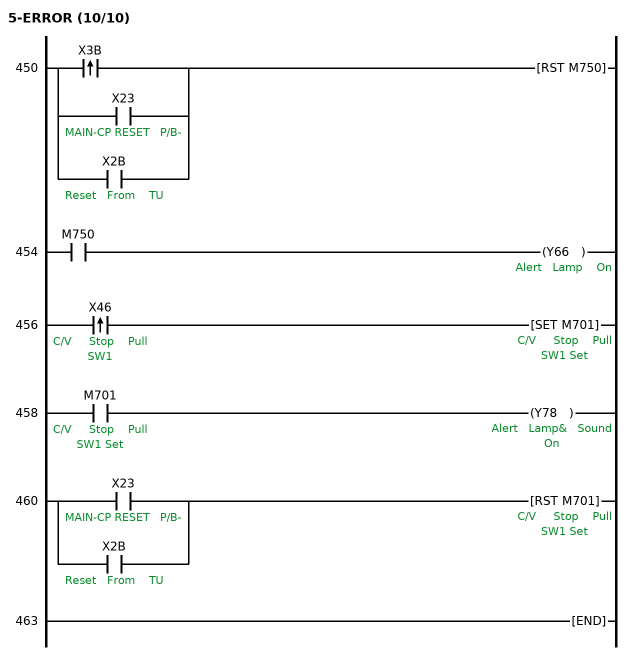
450   LDP     X3B
      OR      X23  ; MAIN-CP RESET   P/B-
      OR      X2B  ; Reset   From    TU
      RST     M750
454   LD      M750
      OUT     Y66  ; Alert   Lamp    On
456   LDP     X46  ; C/V     Stop    Pull    SW1
      SET     M701  ; C/V     Stop    Pull    SW1 Set
458   LD      M701  ; C/V     Stop    Pull    SW1 Set
      OUT     Y78  ; Alert   Lamp&   Sound   On
460   LD      X23  ; MAIN-CP RESET   P/B-
      OR      X2B  ; Reset   From    TU
      RST     M701  ; C/V     Stop    Pull    SW1 Set
463   END
END_PROGRAM

PROGRAM MAIN
0     END
END_PROGRAM

PROGRAM SERVO
